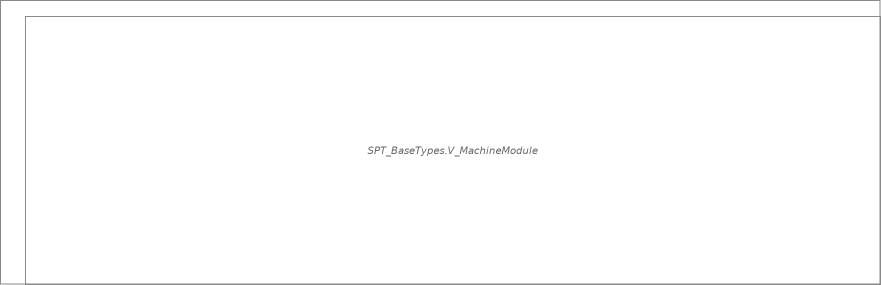
VISUALIZATION Visualization  // 881x285
    Frame (25,16 856x269)
        shows SPT_BaseTypes.V_MachineModule(HMI := MAIN.Machine.PackMLBaseModule_HMI)
END_VISUALIZATION

(* stored: Version 1.1.0.1
   Visu Visualization: Id {a3664553-b48e-4e5a-9724-ae6fd5d8d571} *)
